// TIA Portal V18 export
FUNCTION_BLOCK "nokButton"   // FB11, FBD
{ S7_Optimized_Access := 'TRUE' }
VERSION : 0.1
// stored: AutoNumber true, IsIECCheckEnabled false, IsRetainMemResEnabled false, MemoryReserve 100, SetENOAutomatically false, UDAEnableTagReadback false
   VAR_INPUT
      I_button : Bool;
   END_VAR
   VAR_OUTPUT
      O_buttonLed : Bool;
   END_VAR
   VAR_IN_OUT
      buttonQue : Int;
   END_VAR
   VAR
      fpBit_button : Bool;
      SR_ButtonActive : Bool;
      fpBit_buttonActive : Bool;
      TO_Non_filter { S7_SetPoint := 'True'} : TON_TIME;
      buttonActive { ExternalAccessible := 'False'; ExternalVisible := 'False'; ExternalWritable := 'False'} : Bool;
   END_VAR
   VAR_TEMP
      fp_buttonActive : Bool;
   END_VAR
   VAR_TEMP   // added for the SCL form of the ladder/FBD networks
      _w1 : Bool;
      _w2 : Bool;
   END_VAR
BEGIN

REGION Network 2
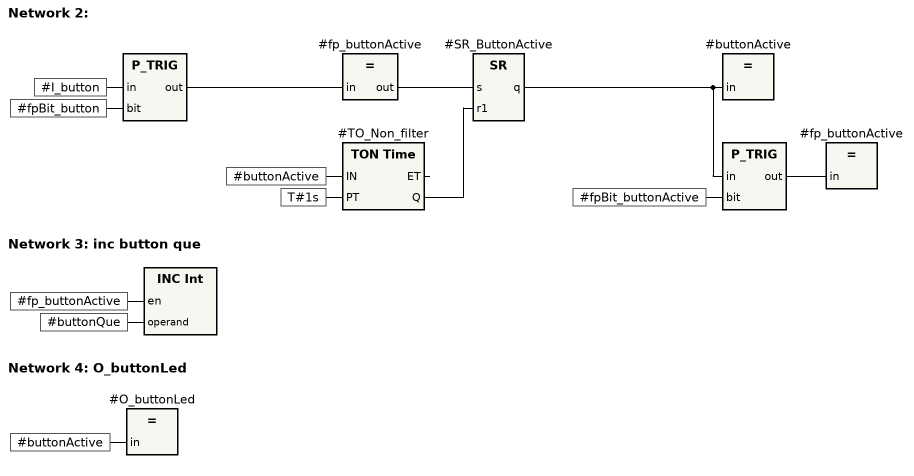
   #_w1 := #I_button AND NOT #fpBit_button;   // rising edge
   #fpBit_button := #I_button;
   #fp_buttonActive := #_w1;
   #TO_Non_filter(IN := #buttonActive, PT := T#1s);   // TON
   IF #_w1 THEN
       #SR_ButtonActive := TRUE;   // SR flip-flop
   END_IF;
   IF #TO_Non_filter.Q THEN #SR_ButtonActive := FALSE; END_IF;
   #buttonActive := #SR_ButtonActive;
   #_w2 := #SR_ButtonActive AND NOT #fpBit_buttonActive;   // rising edge
   #fpBit_buttonActive := #SR_ButtonActive;
   #fp_buttonActive := #_w2;
END_REGION

REGION Network 3: inc button que
   IF #fp_buttonActive THEN #buttonQue := #buttonQue + 1; END_IF;
END_REGION

REGION Network 4: O_buttonLed
   #O_buttonLed := #buttonActive;
END_REGION
END_FUNCTION_BLOCK
